FUNCTION_BLOCK SetParams1Word_DEMUX (* Composite FB wrapping other FBs *)
  (* Standard: 61499-2 *)
  (* Version 1.0, 2021-10-04, dorofeev *)
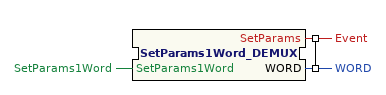
  EVENT_OUTPUT
    SetParams WITH WORD; (* Execution Confirmation *)
  END_EVENT
  VAR_OUTPUT
    WORD : WORD; (* Output event qualifier *)
  END_VAR
  SOCKETS
    SetParams1Word : SetParams1Word;
  END_SOCKETS
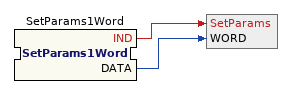
  EVENT_CONNECTIONS
    SetParams1Word.IND TO SetParams;
  END_CONNECTIONS
  DATA_CONNECTIONS
    SetParams1Word.DATA TO WORD;
  END_CONNECTIONS
END_FUNCTION_BLOCK
